{attribute 'GeneratedUsingTerminal: EM3702-0000-0016'}
{attribute addProperty BoxType "EM3702-0000-0016"}
{attribute addProperty Id "AI_Input_Channel_1AT %I*AI_Input_Channel_5AF6604E8AI_Input_Channel_2AT %I*AI_Input_Channel_5AF6604E8WcStateAT %I*WcState_9091E0EB2InfoDataAT %I*InfoData_94A18F5E2"}
{attribute addProperty CRC "3790314305"}
{attribute addProperty Size "20"}
TYPE EM3702_E1EB9B41 EXTENDS EtcSlaveTerminalBase_947E5A46 :
STRUCT
	{attribute addProperty Name "AI_Input_Channel_1"}
	AI_Input_Channel_1 : AI_Input_Channel_5AF6604E;
	{attribute addProperty Name "AI_Input_Channel_2"}
	AI_Input_Channel_2 : AI_Input_Channel_5AF6604E;
	{attribute addProperty Name "WcState"}
	WcState : WcState_9091E0EB;
	{attribute addProperty Name "InfoData"}
	InfoData : InfoData_94A18F5E;
END_STRUCT
END_TYPE

(* stored: Version 1.2.0.0, ProductVersion 3.1.4024.9
   DUT EM3702_E1EB9B41: Id {3bc4e7df-f793-4c43-9a42-dfbf11c1e0c3} *)
